{attribute 'qualified_only'}
VAR_GLOBAL
	TR_P2_WT2_rValue_REAL: REAL;
END_VAR

(* stored: Version 1.1.0.1, ProductVersion 3.1.4024.14
   GVL CanOpen: Id {19b84136-68f9-482b-b40f-687f26e5e121} *)
